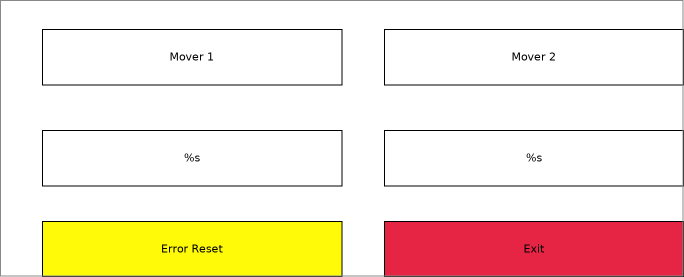
VISUALIZATION Settings  // 684x277
    RoundedRectangle (42,29 300x56), "Mover 1"
    RoundedRectangle (42,130 300x56), "%s", text variable: MAIN.stMoverState
        p4168582468: MAIN.stMoverState
    RoundedRectangle (384,29 300x56), "Mover 2"
    RoundedRectangle (384,130 300x56), "%s", text variable: MAIN.stMoverState2
    RoundedRectangle (42,221 300x56), "Error Reset"
        tap MAIN.bReset
    RoundedRectangle (384,221 300x56), "Exit"
        OnMouseClick: change screen: RaceControls
END_VISUALIZATION

(* stored: Version 1.1.0.1
   Visu Settings: Id {0bdcac43-6a04-4985-87fe-927afbfdc9fb} *)
